(* CODESYS project FIO.export

Project tree, tasks and I/O mapping:
  global variables FIO
*)

// FIO
{attribute 'qualified_only'}
VAR_GLOBAL
	(*Inputs*)
    iAtEntry        : BOOL;
    iLowBox         : BOOL;
    iHighBox        : BOOL;
    iAtTurnEntry    : BOOL;
    iAtLoadPos      : BOOL;
    iAtUnloadPos    : BOOL;
    iAtFront        : BOOL;
    iAtRightEntry   : BOOL;
    iAtLeftEntry    : BOOL;
    iAtRightExit    : BOOL;
    iAtLeftExit     : BOOL;
	
	iStart			: BOOL;
	iStop			: BOOL;
	iReset			: BOOL;
	iManual			: BOOL;
	iAuto			: BOOL;
	iEmergencyStop	: BOOL;
	
	(*Outputs*)
    oFeederConveyor : BOOL;
    oEntryConveyor  : BOOL;
    oLoad           : BOOL;
    oUnload         : BOOL;
    oTurn           : BOOL;
    oLeftConveyor   : BOOL;
    oRightConveyor  : BOOL;
	
	oStartLight		: BOOL;
	oStopLight		: BOOL;
	oResetLight		: BOOL;
	ointCounter		: INT;
	ointTest		:INT;
	
	
	oGreenIndicator	: BOOL;
	oRedIndicator	: BOOL;
	oYellowIndicator : BOOL;
	
	(*HMI Buttons*)
	buttonFeederConveyor : BOOL;
    buttonEntryConveyor  : BOOL;
    buttonLoad           : BOOL;
    buttonUnload         : BOOL;
    buttonTurn           : BOOL;
    buttonLeftConveyor   : BOOL;
    buttonRightConveyor  : BOOL;
	
	
END_VAR
